{attribute 'linkalways'} 
{attribute 'no_explicit_call' := 'This FB is a CLASS and must be accessed using methods or properties'}
{attribute 'enable_dynamic_creation'}
FUNCTION_BLOCK MockEnumDatatype_E_TcEventClass EXTENDS EnumDatatypeBase
VAR
	localData : E_TcEventClass;
	activeData : REFERENCE TO E_TcEventClass;
	enumBaseDatatype : _UINT(localData);
END_VAR

METHOD PRIVATE AddLocalEnumeration
VAR_INPUT
	Enumeration : T_MAXSTRING;
	Value : E_TcEventClass;
END_VAR
AddEnumeration(Enumeration, Value);
END_METHOD

PROPERTY PUBLIC Address : PVOID
GET
Address := ADR(activeData);
END_GET
END_PROPERTY

METHOD PUBLIC ClearReference
VAR_INPUT
END_VAR
activeData REF= localData;
SetBaseDatatypeReference();
END_METHOD

METHOD PUBLIC Clone : I_Datatype
VAR
    pClone : POINTER TO MockEnumDatatype_E_TcEventClass;
END_VAR
pClone := __NEW(MockEnumDatatype_E_TcEventClass(InitialValue := Value));
Clone := pClone^;
END_METHOD

METHOD FB_init : BOOL
VAR_INPUT
	bInitRetains : BOOL; // if TRUE, the retain variables are initialized (warm start / cold start)
	bInCopyCode : BOOL;  // if TRUE, the instance afterwards gets moved into the copy code (online change)
	InitialValue : E_TcEventClass;
END_VAR
localData := InitialValue;
AddBaseDatatype(enumBaseDatatype);
ClearReference();

AddLocalEnumeration('TCEVENTCLASS_NONE', E_TcEventClass.TCEVENTCLASS_NONE);
AddLocalEnumeration('TCEVENTCLASS_MAINTENANCE', E_TcEventClass.TCEVENTCLASS_MAINTENANCE);
AddLocalEnumeration('TCEVENTCLASS_MESSAGE', E_TcEventClass.TCEVENTCLASS_MESSAGE);
AddLocalEnumeration('TCEVENTCLASS_HINT', E_TcEventClass.TCEVENTCLASS_HINT);
AddLocalEnumeration('TCEVENTCLASS_STATEINFO', E_TcEventClass.TCEVENTCLASS_STATEINFO);
AddLocalEnumeration('TCEVENTCLASS_INSTRUCTION', E_TcEventClass.TCEVENTCLASS_INSTRUCTION);
AddLocalEnumeration('TCEVENTCLASS_WARNING', E_TcEventClass.TCEVENTCLASS_WARNING);
AddLocalEnumeration('TCEVENTCLASS_ALARM', E_TcEventClass.TCEVENTCLASS_ALARM);
AddLocalEnumeration('TCEVENTCLASS_PARAMERROR', E_TcEventClass.TCEVENTCLASS_PARAMERROR);
END_METHOD

PROPERTY PUBLIC Identifier : T_MAXSTRING
GET
Identifier := 'E_TcEventClass';
END_GET
END_PROPERTY

METHOD IsEnumeratorValueEqual : BOOL
VAR_INPUT
	Enumerator : I_KeyValueForwardEnumerator;
END_VAR
VAR
	storedValue : E_TcEventClass;
END_VAR
IF NOT Enumerator.TryGet(storedValue) THEN
	RETURN;
END_IF

IsEnumeratorValueEqual := storedValue = activeData;
END_METHOD

METHOD PUBLIC MakeReferenceTo
VAR_INPUT
	ReferenceTarget : REFERENCE TO E_TcEventClass;
END_VAR
activeData REF= ReferenceTarget;
SetBaseDatatypeReference();
END_METHOD

METHOD PROTECTED SetBaseDatatypeReference
VAR_INPUT
END_VAR
enumBaseDatatype.MakeReferenceTo(activeData);
END_METHOD

PROPERTY PUBLIC Size : UDINT
GET
Size := SIZEOF(activeData);
END_GET
END_PROPERTY

METHOD TryMakeReferenceTo : BOOL
VAR_INPUT
	Target : I_Datatype;
END_VAR
VAR
	targetAsEnum : I_EnumDatatype;
	pTargetData : POINTER TO E_TcEventClass;
END_VAR
IF NOT Target.TryResolveAsEnumDatatype(targetAsEnum) THEN
	RETURN;
END_IF

IF targetAsEnum.Identifier <> Identifier THEN
	RETURN;
END_IF

pTargetData := Target.Address;
activeData REF= pTargetData^;
SetBaseDatatypeReference();
TryMakeReferenceTo := TRUE;
END_METHOD

PROPERTY PUBLIC Value : E_TcEventClass
GET
Value := activeData;
END_GET
SET
activeData := Value;
END_SET
END_PROPERTY

END_FUNCTION_BLOCK

(* stored: Version 1.1.0.1, ProductVersion 3.1.4024.12
   POU MockEnumDatatype_E_TcEventClass: Id {5be12e34-c0d1-4973-8284-039090e83858}, SpecialFunc None
   Folder Constructor: Id {72c73cd4-5112-4575-a4ce-4926caae75c4}
   Folder Private: Id {f64647d7-c4ad-474a-a85a-418458d7d9d6}
   Folder Protected: Id {10fad48b-6bbf-400a-b933-52ef692221ce}
   Method AddLocalEnumeration: Id {52effdbd-37fa-453c-baa2-8882527e3912}
   Property Address: Id {dc25011f-b2a0-4420-98c8-b921c98f340c}
   Get Get: Id {66625fcb-a0fd-4385-9e81-d11485dab810}
   Method ClearReference: Id {7b147035-0843-456a-b403-3f67350949d6}
   Method Clone: Id {77d4e1ef-06b6-459a-9194-edbcd6394657}
   Method FB_init: Id {8ef90484-7f12-4187-94f2-3b44a21100d9}
   Property Identifier: Id {5342fd20-72dc-444d-a214-55c0dd5ad52c}
   Get Get: Id {56fc425c-b7ce-4e6e-b6d1-aa9af0d39f1d}
   Method IsEnumeratorValueEqual: Id {6a61e91c-9236-46f1-8155-81d72ee95224}
   Method MakeReferenceTo: Id {646f68ea-4df1-4b73-bffa-1a01bba19e03}
   Method SetBaseDatatypeReference: Id {130acbcc-f84e-4ae1-8b25-95d6d588f69a}
   Property Size: Id {57f25cab-adc7-44a6-8f0a-6f08ed25c722}
   Get Get: Id {929cef7a-424d-4d36-8027-fe9020dc4298}
   Method TryMakeReferenceTo: Id {ce5f5830-b861-40e9-8958-4ad17ed78f1e}
   Property Value: Id {bee402f6-2aca-40e1-a610-51bc94e1ddb1}
   Get Get: Id {56ecd470-c691-43cd-bcf4-03ab287375cd}
   Set Set: Id {bc022720-64b4-4688-888a-494ca5f6e0c4} *)
